Staubli VAL3: getLibVersion.pgx

public program getLibVersion(string& version_[])
begin
  // retrieve version of library
  version_=strVersion
end
